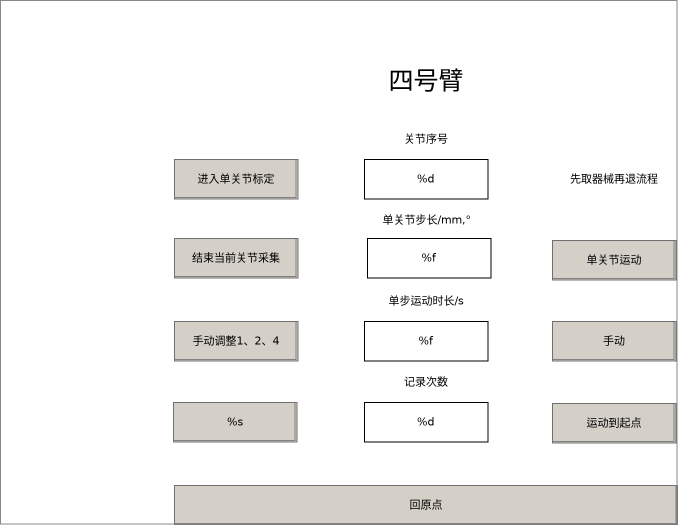
VISUALIZATION kineCali_a4  // 678x525
    Button (174,159 124x40), "进入单关节标定", colour toggle: g_singleJntTest.m_enterSingleJntTestMode[4]
        toggle g_singleJntTest.m_enterSingleJntTestMode[4]
    Button (552,321 124x40), "手动", colour toggle: g_singleJntTest.m_manualAdjustFlag
    Button (552,403 124x40), "运动到起点", colour toggle: g_singleJntTest.m_move2StartFlag
    Rectangle (364,402 124x40), "%d", text variable: g_singleJntTest.m_dataRecordCount[4]
        OnMouseClick: write the text variable via Default, min 0, max 1000
    Label (352,200 150x40), "单关节步长/mm,°"
    Button (552,240 124x40), "单关节运动", colour toggle: g_singleJntTest.m_singleJntFlag
    Label (351,119 150x40), "关节序号"
    Rectangle (367,238 124x40), "%f", text variable: g_singleJntTest.m_jntStep
        OnMouseClick: write the text variable via Default, min 0
    Button (173,402 124x40), "%s", text variable: g_singleJntTest.m_dataRecordText, colour toggle: g_singleJntTest.m_dataRecordFlag[4]
        tap g_singleJntTest.m_dataRecordFlag[4]
    Rectangle (364,159 124x40), "%d", text variable: g_singleJntTest.m_kineCaliJntIdx
        OnMouseClick: write the text variable via Default, min 1, max 8
    Button (174,485 504x40), "回原点", colour toggle: g_singleJntTest.m_return2OriginFlag
        toggle g_singleJntTest.m_return2OriginFlag
    Rectangle (364,321 124x40), "%f", text variable: g_singleJntTest.m_EndT
        OnMouseClick: write the text variable via Default, min 0, max 100
    Label (351,281 150x40), "单步运动时长/s"
    Label (351,362 150x40), "记录次数"
    Label (351,59 150x43), "四号臂"
    Button (174,238 124x40), "结束当前关节采集", colour toggle: g_singleJntTest.m_manualEndFlag
        toggle g_singleJntTest.m_manualEndFlag
    Button (174,321 124x40), "手动调整1、2、4", colour toggle: g_singleJntTest.m_manual124StartFlag
        toggle g_singleJntTest.m_manual124StartFlag
    Label (552,159 124x40), "先取器械再退流程"
END_VISUALIZATION

(* stored: Version 1.1.0.1, ProductVersion 3.1.4024.11
   Visu kineCali_a4: Id {abbd2810-91b7-4230-a7d0-f3cfd191b78d} *)
